// TIA Portal V15.1 export
// export: Created 2026-01-15T16:29:41.881654Z, ExportSetting WithDefaults, WithReadOnly, DisplayName Totally Integrated Automation Portal, DisplayVersion V15.1 Update 8, DisplayName TIA Portal Openness, DisplayVersion V15.1 Update 8, DisplayName STEP 7 Professional, DisplayVersion V15.1 Update 8, DisplayName WinCC Advanced, DisplayVersion V15.1 Update 8
FUNCTION_BLOCK "4.SIMULATION_DATA"   // FB4, LAD
{ S7_Optimized_Access := 'TRUE' }
VERSION : 0.1
// stored: AutoNumber false, CodeModifiedDate 2025-08-27T17:12:03.7644125Z, CompileDate 2026-01-15T16:25:51.5973447Z, CreationDate 2026-01-15T16:22:49.8270549Z, DownloadWithoutReinit false, HandleErrorsWithinBlock false, InterfaceModifiedDate 2023-11-28T22:28:44.2264332Z, IsConsistent true, IsIECCheckEnabled false, IsKnowHowProtected false, IsRetainMemResEnabled false, IsWriteProtected false, LibraryConformanceStatus The object is library-conformant., MemoryReserve 100, ModifiedDate 2025-08-27T17:12:03.7644125Z, ParameterModified 2023-11-28T22:28:44.2264332Z, PLCSimAdvancedSupport false, SetENOAutomatically False, StructureModified 2023-11-28T22:28:44.2264332Z, UDAEnableTagReadback false
   VAR_INPUT
      RE_SET : Bool;
      XUNG_CLOCK : Bool;
      CAN_1 : Bool;
      CAN_2 : Bool;
      CAN_3 : Bool;
      CAN_4 : Bool;
      CAN_5 : Bool;
      CAN_6 : Bool;
      CAN_7 : Bool;
      CAN_8 : Bool;
      CAN_9 : Bool;
      CAN_10 : Bool;
      CAN_11 : Bool;
      CAN_12 : Bool;
      XA_1 : Bool;
      XA_2 : Bool;
      XA_3 : Bool;
      XA_4 : Bool;
      XA_5 : Bool;
      XA_6 : Bool;
      XA_7 : Bool;
      XA_8 : Bool;
      XA_9 : Bool;
      XA_10 : Bool;
      XA_11 : Bool;
      XA_12 : Bool;
      HS_NAP_AGG1 : Real;
      HS_NAP_AGG2 : Real;
      HS_NAP_AGG3 : Real;
      HS_NAP_AGG4 : Real;
      HS_NAP_AGG5 : Real;
      HS_NAP_AGG6 : Real;
      HS_NAP_CEM1 : Real;
      HS_NAP_CEM2 : Real;
      HS_NAP_WAT1 : Real;
      HS_NAP_WAT2 : Real;
      HS_NAP_ADD1 : Real;
      HS_NAP_ADD2 : Real;
      HS_XA_AGG1 : Real;
      HS_XA_AGG2 : Real;
      HS_XA_AGG3 : Real;
      HS_XA_AGG4 : Real;
      HS_XA_AGG5 : Real;
      HS_XA_AGG6 : Real;
      HS_XA_CEM1 : Real;
      HS_XA_CEM2 : Real;
      HS_XA_WAT1 : Real;
      HS_XA_WAT2 : Real;
      HS_XA_ADD1 : Real;
      HS_XA_ADD2 : Real;
   END_VAR
   VAR_OUTPUT
      AGG1 : Real;
      AGG2 : Real;
      AGG3 : Real;
      AGG4 : Real;
      AGG5 : Real;
      AGG6 : Real;
      CEM1 : Real;
      CEM2 : Real;
      WAT1 : Real;
      WAT2 : Real;
      WADD1 : Real;
      WADD2 : Real;
   END_VAR
   VAR
      A1 : Bool;
      B1 : Bool;
      A2 : Bool;
      B2 : Bool;
      A3 : Bool;
      B3 : Bool;
      A4 : Bool;
      B4 : Bool;
      A5 : Bool;
      B5 : Bool;
      A6 : Bool;
      B6 : Bool;
      A7 : Bool;
      B7 : Bool;
      A8 : Bool;
      B8 : Bool;
      A9 : Bool;
      B9 : Bool;
      A10 : Bool;
      B10 : Bool;
      A11 : Bool;
      B11 : Bool;
      A12 : Bool;
      B12 : Bool;
   END_VAR
   VAR_TEMP   // added for the SCL form of the ladder/FBD networks
      _w1 : Bool;
      _w2 : Bool;
   END_VAR
BEGIN

REGION Network 1: RESET
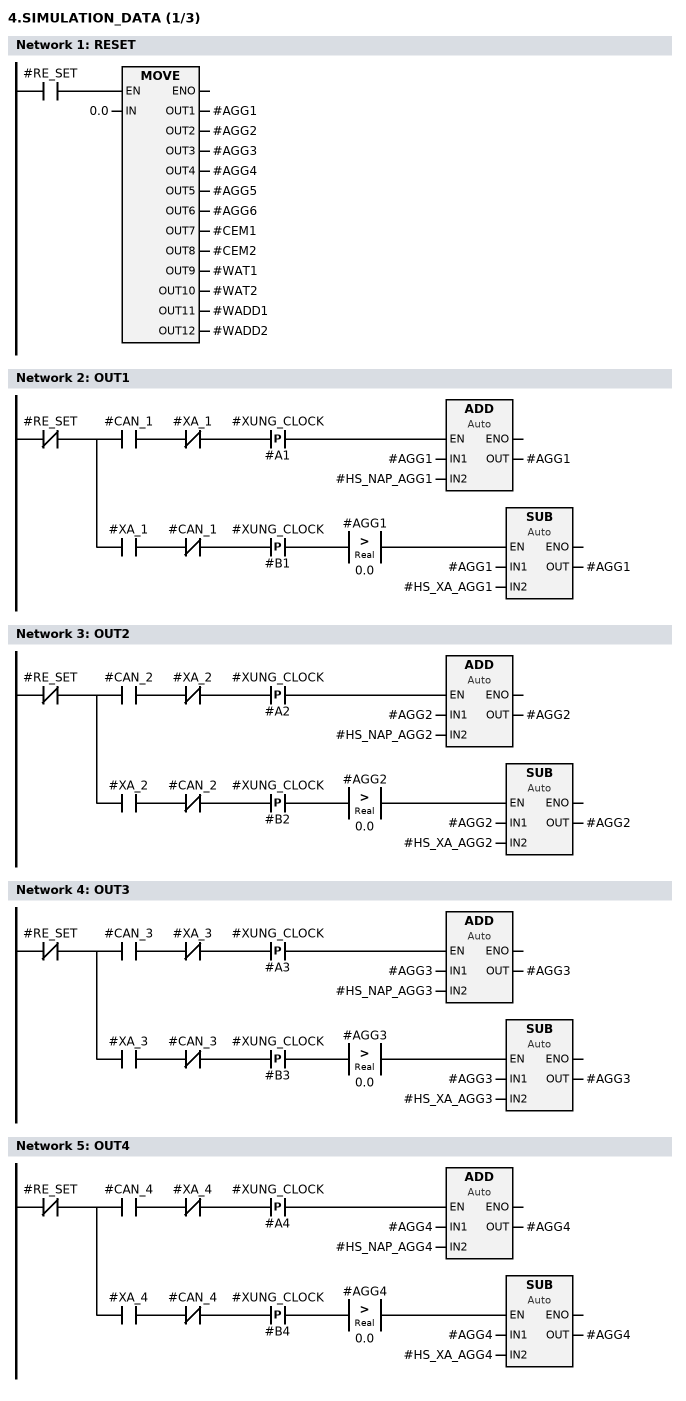
   RUNG wire#powerrail
      Contact( #RE_SET )
      Move(in := 0.0, out1 => #AGG1, out2 => #AGG2, out3 => #AGG3, out4 => #AGG4, out5 => #AGG5, out6 => #AGG6, out7 => #CEM1, out8 => #CEM2, out9 => #WAT1, out10 => #WAT2, out11 => #WADD1, out12 => #WADD2)
   END_RUNG
   // the same network as SCL:
   IF #RE_SET THEN
       #AGG1 := 0.0;
       #AGG2 := 0.0;
       #AGG3 := 0.0;
       #AGG4 := 0.0;
       #AGG5 := 0.0;
       #AGG6 := 0.0;
       #CEM1 := 0.0;
       #CEM2 := 0.0;
       #WAT1 := 0.0;
       #WAT2 := 0.0;
       #WADD1 := 0.0;
       #WADD2 := 0.0;
   END_IF;
END_REGION

REGION Network 2: OUT1
   RUNG wire#powerrail
      I_Contact( #RE_SET )
      wire#w1
      Contact( #CAN_1 )
      I_Contact( #XA_1 )
      P_Contact(operand := #XUNG_CLOCK, bit := #A1)
      Add(in1 := #AGG1, in2 := #HS_NAP_AGG1, out => #AGG1)
   END_RUNG
   RUNG wire#w1
      Contact( #XA_1 )
      I_Contact( #CAN_1 )
      P_Contact(operand := #XUNG_CLOCK, bit := #B1)
      { S7_Templates := "SrcType := Real" } GT_Contact(in1 := #AGG1, in2 := 0.0)
      Sub(in1 := #AGG1, in2 := #HS_XA_AGG1, out => #AGG1)
   END_RUNG
   // the same network as SCL:
   #_w1 := NOT #RE_SET AND #CAN_1 AND NOT #XA_1 AND #XUNG_CLOCK AND NOT #A1;   // rising edge of #XUNG_CLOCK
   #A1 := #XUNG_CLOCK;
   IF #_w1 THEN #AGG1 := #AGG1 + #HS_NAP_AGG1; END_IF;
   #_w2 := NOT #RE_SET AND #XA_1 AND NOT #CAN_1 AND #XUNG_CLOCK AND NOT #B1;   // rising edge of #XUNG_CLOCK
   #B1 := #XUNG_CLOCK;
   IF #_w2 AND (#AGG1 > 0.0) THEN #AGG1 := #AGG1 - #HS_XA_AGG1; END_IF;
END_REGION

REGION Network 3: OUT2
   RUNG wire#powerrail
      I_Contact( #RE_SET )
      wire#w1
      Contact( #CAN_2 )
      I_Contact( #XA_2 )
      P_Contact(operand := #XUNG_CLOCK, bit := #A2)
      Add(in1 := #AGG2, in2 := #HS_NAP_AGG2, out => #AGG2)
   END_RUNG
   RUNG wire#w1
      Contact( #XA_2 )
      I_Contact( #CAN_2 )
      P_Contact(operand := #XUNG_CLOCK, bit := #B2)
      { S7_Templates := "SrcType := Real" } GT_Contact(in1 := #AGG2, in2 := 0.0)
      Sub(in1 := #AGG2, in2 := #HS_XA_AGG2, out => #AGG2)
   END_RUNG
   // the same network as SCL:
   #_w1 := NOT #RE_SET AND #CAN_2 AND NOT #XA_2 AND #XUNG_CLOCK AND NOT #A2;   // rising edge of #XUNG_CLOCK
   #A2 := #XUNG_CLOCK;
   IF #_w1 THEN #AGG2 := #AGG2 + #HS_NAP_AGG2; END_IF;
   #_w2 := NOT #RE_SET AND #XA_2 AND NOT #CAN_2 AND #XUNG_CLOCK AND NOT #B2;   // rising edge of #XUNG_CLOCK
   #B2 := #XUNG_CLOCK;
   IF #_w2 AND (#AGG2 > 0.0) THEN #AGG2 := #AGG2 - #HS_XA_AGG2; END_IF;
END_REGION

REGION Network 4: OUT3
   RUNG wire#powerrail
      I_Contact( #RE_SET )
      wire#w1
      Contact( #CAN_3 )
      I_Contact( #XA_3 )
      P_Contact(operand := #XUNG_CLOCK, bit := #A3)
      Add(in1 := #AGG3, in2 := #HS_NAP_AGG3, out => #AGG3)
   END_RUNG
   RUNG wire#w1
      Contact( #XA_3 )
      I_Contact( #CAN_3 )
      P_Contact(operand := #XUNG_CLOCK, bit := #B3)
      { S7_Templates := "SrcType := Real" } GT_Contact(in1 := #AGG3, in2 := 0.0)
      Sub(in1 := #AGG3, in2 := #HS_XA_AGG3, out => #AGG3)
   END_RUNG
   // the same network as SCL:
   #_w1 := NOT #RE_SET AND #CAN_3 AND NOT #XA_3 AND #XUNG_CLOCK AND NOT #A3;   // rising edge of #XUNG_CLOCK
   #A3 := #XUNG_CLOCK;
   IF #_w1 THEN #AGG3 := #AGG3 + #HS_NAP_AGG3; END_IF;
   #_w2 := NOT #RE_SET AND #XA_3 AND NOT #CAN_3 AND #XUNG_CLOCK AND NOT #B3;   // rising edge of #XUNG_CLOCK
   #B3 := #XUNG_CLOCK;
   IF #_w2 AND (#AGG3 > 0.0) THEN #AGG3 := #AGG3 - #HS_XA_AGG3; END_IF;
END_REGION

REGION Network 5: OUT4
   RUNG wire#powerrail
      I_Contact( #RE_SET )
      wire#w1
      Contact( #CAN_4 )
      I_Contact( #XA_4 )
      P_Contact(operand := #XUNG_CLOCK, bit := #A4)
      Add(in1 := #AGG4, in2 := #HS_NAP_AGG4, out => #AGG4)
   END_RUNG
   RUNG wire#w1
      Contact( #XA_4 )
      I_Contact( #CAN_4 )
      P_Contact(operand := #XUNG_CLOCK, bit := #B4)
      { S7_Templates := "SrcType := Real" } GT_Contact(in1 := #AGG4, in2 := 0.0)
      Sub(in1 := #AGG4, in2 := #HS_XA_AGG4, out => #AGG4)
   END_RUNG
   // the same network as SCL:
   #_w1 := NOT #RE_SET AND #CAN_4 AND NOT #XA_4 AND #XUNG_CLOCK AND NOT #A4;   // rising edge of #XUNG_CLOCK
   #A4 := #XUNG_CLOCK;
   IF #_w1 THEN #AGG4 := #AGG4 + #HS_NAP_AGG4; END_IF;
   #_w2 := NOT #RE_SET AND #XA_4 AND NOT #CAN_4 AND #XUNG_CLOCK AND NOT #B4;   // rising edge of #XUNG_CLOCK
   #B4 := #XUNG_CLOCK;
   IF #_w2 AND (#AGG4 > 0.0) THEN #AGG4 := #AGG4 - #HS_XA_AGG4; END_IF;
END_REGION

REGION Network 6: OUT5
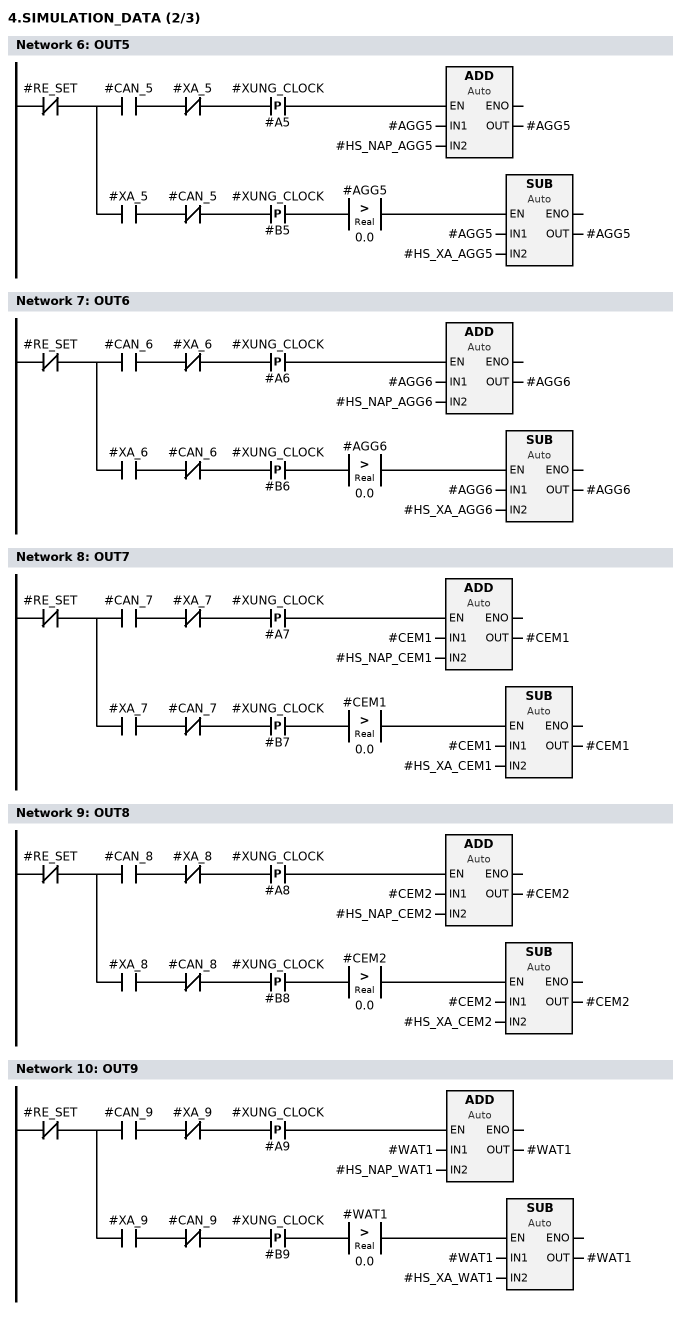
   RUNG wire#powerrail
      I_Contact( #RE_SET )
      wire#w1
      Contact( #CAN_5 )
      I_Contact( #XA_5 )
      P_Contact(operand := #XUNG_CLOCK, bit := #A5)
      Add(in1 := #AGG5, in2 := #HS_NAP_AGG5, out => #AGG5)
   END_RUNG
   RUNG wire#w1
      Contact( #XA_5 )
      I_Contact( #CAN_5 )
      P_Contact(operand := #XUNG_CLOCK, bit := #B5)
      { S7_Templates := "SrcType := Real" } GT_Contact(in1 := #AGG5, in2 := 0.0)
      Sub(in1 := #AGG5, in2 := #HS_XA_AGG5, out => #AGG5)
   END_RUNG
   // the same network as SCL:
   #_w1 := NOT #RE_SET AND #CAN_5 AND NOT #XA_5 AND #XUNG_CLOCK AND NOT #A5;   // rising edge of #XUNG_CLOCK
   #A5 := #XUNG_CLOCK;
   IF #_w1 THEN #AGG5 := #AGG5 + #HS_NAP_AGG5; END_IF;
   #_w2 := NOT #RE_SET AND #XA_5 AND NOT #CAN_5 AND #XUNG_CLOCK AND NOT #B5;   // rising edge of #XUNG_CLOCK
   #B5 := #XUNG_CLOCK;
   IF #_w2 AND (#AGG5 > 0.0) THEN #AGG5 := #AGG5 - #HS_XA_AGG5; END_IF;
END_REGION

REGION Network 7: OUT6
   RUNG wire#powerrail
      I_Contact( #RE_SET )
      wire#w1
      Contact( #CAN_6 )
      I_Contact( #XA_6 )
      P_Contact(operand := #XUNG_CLOCK, bit := #A6)
      Add(in1 := #AGG6, in2 := #HS_NAP_AGG6, out => #AGG6)
   END_RUNG
   RUNG wire#w1
      Contact( #XA_6 )
      I_Contact( #CAN_6 )
      P_Contact(operand := #XUNG_CLOCK, bit := #B6)
      { S7_Templates := "SrcType := Real" } GT_Contact(in1 := #AGG6, in2 := 0.0)
      Sub(in1 := #AGG6, in2 := #HS_XA_AGG6, out => #AGG6)
   END_RUNG
   // the same network as SCL:
   #_w1 := NOT #RE_SET AND #CAN_6 AND NOT #XA_6 AND #XUNG_CLOCK AND NOT #A6;   // rising edge of #XUNG_CLOCK
   #A6 := #XUNG_CLOCK;
   IF #_w1 THEN #AGG6 := #AGG6 + #HS_NAP_AGG6; END_IF;
   #_w2 := NOT #RE_SET AND #XA_6 AND NOT #CAN_6 AND #XUNG_CLOCK AND NOT #B6;   // rising edge of #XUNG_CLOCK
   #B6 := #XUNG_CLOCK;
   IF #_w2 AND (#AGG6 > 0.0) THEN #AGG6 := #AGG6 - #HS_XA_AGG6; END_IF;
END_REGION

REGION Network 8: OUT7
   RUNG wire#powerrail
      I_Contact( #RE_SET )
      wire#w1
      Contact( #CAN_7 )
      I_Contact( #XA_7 )
      P_Contact(operand := #XUNG_CLOCK, bit := #A7)
      Add(in1 := #CEM1, in2 := #HS_NAP_CEM1, out => #CEM1)
   END_RUNG
   RUNG wire#w1
      Contact( #XA_7 )
      I_Contact( #CAN_7 )
      P_Contact(operand := #XUNG_CLOCK, bit := #B7)
      { S7_Templates := "SrcType := Real" } GT_Contact(in1 := #CEM1, in2 := 0.0)
      Sub(in1 := #CEM1, in2 := #HS_XA_CEM1, out => #CEM1)
   END_RUNG
   // the same network as SCL:
   #_w1 := NOT #RE_SET AND #CAN_7 AND NOT #XA_7 AND #XUNG_CLOCK AND NOT #A7;   // rising edge of #XUNG_CLOCK
   #A7 := #XUNG_CLOCK;
   IF #_w1 THEN #CEM1 := #CEM1 + #HS_NAP_CEM1; END_IF;
   #_w2 := NOT #RE_SET AND #XA_7 AND NOT #CAN_7 AND #XUNG_CLOCK AND NOT #B7;   // rising edge of #XUNG_CLOCK
   #B7 := #XUNG_CLOCK;
   IF #_w2 AND (#CEM1 > 0.0) THEN #CEM1 := #CEM1 - #HS_XA_CEM1; END_IF;
END_REGION

REGION Network 9: OUT8
   RUNG wire#powerrail
      I_Contact( #RE_SET )
      wire#w1
      Contact( #CAN_8 )
      I_Contact( #XA_8 )
      P_Contact(operand := #XUNG_CLOCK, bit := #A8)
      Add(in1 := #CEM2, in2 := #HS_NAP_CEM2, out => #CEM2)
   END_RUNG
   RUNG wire#w1
      Contact( #XA_8 )
      I_Contact( #CAN_8 )
      P_Contact(operand := #XUNG_CLOCK, bit := #B8)
      { S7_Templates := "SrcType := Real" } GT_Contact(in1 := #CEM2, in2 := 0.0)
      Sub(in1 := #CEM2, in2 := #HS_XA_CEM2, out => #CEM2)
   END_RUNG
   // the same network as SCL:
   #_w1 := NOT #RE_SET AND #CAN_8 AND NOT #XA_8 AND #XUNG_CLOCK AND NOT #A8;   // rising edge of #XUNG_CLOCK
   #A8 := #XUNG_CLOCK;
   IF #_w1 THEN #CEM2 := #CEM2 + #HS_NAP_CEM2; END_IF;
   #_w2 := NOT #RE_SET AND #XA_8 AND NOT #CAN_8 AND #XUNG_CLOCK AND NOT #B8;   // rising edge of #XUNG_CLOCK
   #B8 := #XUNG_CLOCK;
   IF #_w2 AND (#CEM2 > 0.0) THEN #CEM2 := #CEM2 - #HS_XA_CEM2; END_IF;
END_REGION

REGION Network 10: OUT9
   RUNG wire#powerrail
      I_Contact( #RE_SET )
      wire#w1
      Contact( #CAN_9 )
      I_Contact( #XA_9 )
      P_Contact(operand := #XUNG_CLOCK, bit := #A9)
      Add(in1 := #WAT1, in2 := #HS_NAP_WAT1, out => #WAT1)
   END_RUNG
   RUNG wire#w1
      Contact( #XA_9 )
      I_Contact( #CAN_9 )
      P_Contact(operand := #XUNG_CLOCK, bit := #B9)
      { S7_Templates := "SrcType := Real" } GT_Contact(in1 := #WAT1, in2 := 0.0)
      Sub(in1 := #WAT1, in2 := #HS_XA_WAT1, out => #WAT1)
   END_RUNG
   // the same network as SCL:
   #_w1 := NOT #RE_SET AND #CAN_9 AND NOT #XA_9 AND #XUNG_CLOCK AND NOT #A9;   // rising edge of #XUNG_CLOCK
   #A9 := #XUNG_CLOCK;
   IF #_w1 THEN #WAT1 := #WAT1 + #HS_NAP_WAT1; END_IF;
   #_w2 := NOT #RE_SET AND #XA_9 AND NOT #CAN_9 AND #XUNG_CLOCK AND NOT #B9;   // rising edge of #XUNG_CLOCK
   #B9 := #XUNG_CLOCK;
   IF #_w2 AND (#WAT1 > 0.0) THEN #WAT1 := #WAT1 - #HS_XA_WAT1; END_IF;
END_REGION

REGION Network 11: OUT10
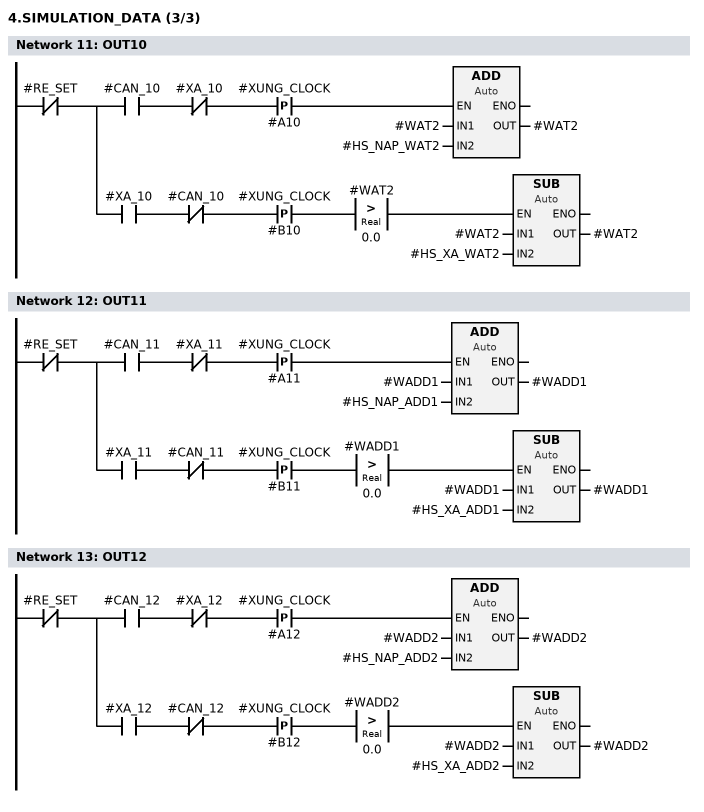
   RUNG wire#powerrail
      I_Contact( #RE_SET )
      wire#w1
      Contact( #CAN_10 )
      I_Contact( #XA_10 )
      P_Contact(operand := #XUNG_CLOCK, bit := #A10)
      Add(in1 := #WAT2, in2 := #HS_NAP_WAT2, out => #WAT2)
   END_RUNG
   RUNG wire#w1
      Contact( #XA_10 )
      I_Contact( #CAN_10 )
      P_Contact(operand := #XUNG_CLOCK, bit := #B10)
      { S7_Templates := "SrcType := Real" } GT_Contact(in1 := #WAT2, in2 := 0.0)
      Sub(in1 := #WAT2, in2 := #HS_XA_WAT2, out => #WAT2)
   END_RUNG
   // the same network as SCL:
   #_w1 := NOT #RE_SET AND #CAN_10 AND NOT #XA_10 AND #XUNG_CLOCK AND NOT #A10;   // rising edge of #XUNG_CLOCK
   #A10 := #XUNG_CLOCK;
   IF #_w1 THEN #WAT2 := #WAT2 + #HS_NAP_WAT2; END_IF;
   #_w2 := NOT #RE_SET AND #XA_10 AND NOT #CAN_10 AND #XUNG_CLOCK AND NOT #B10;   // rising edge of #XUNG_CLOCK
   #B10 := #XUNG_CLOCK;
   IF #_w2 AND (#WAT2 > 0.0) THEN #WAT2 := #WAT2 - #HS_XA_WAT2; END_IF;
END_REGION

REGION Network 12: OUT11
   RUNG wire#powerrail
      I_Contact( #RE_SET )
      wire#w1
      Contact( #CAN_11 )
      I_Contact( #XA_11 )
      P_Contact(operand := #XUNG_CLOCK, bit := #A11)
      Add(in1 := #WADD1, in2 := #HS_NAP_ADD1, out => #WADD1)
   END_RUNG
   RUNG wire#w1
      Contact( #XA_11 )
      I_Contact( #CAN_11 )
      P_Contact(operand := #XUNG_CLOCK, bit := #B11)
      { S7_Templates := "SrcType := Real" } GT_Contact(in1 := #WADD1, in2 := 0.0)
      Sub(in1 := #WADD1, in2 := #HS_XA_ADD1, out => #WADD1)
   END_RUNG
   // the same network as SCL:
   #_w1 := NOT #RE_SET AND #CAN_11 AND NOT #XA_11 AND #XUNG_CLOCK AND NOT #A11;   // rising edge of #XUNG_CLOCK
   #A11 := #XUNG_CLOCK;
   IF #_w1 THEN #WADD1 := #WADD1 + #HS_NAP_ADD1; END_IF;
   #_w2 := NOT #RE_SET AND #XA_11 AND NOT #CAN_11 AND #XUNG_CLOCK AND NOT #B11;   // rising edge of #XUNG_CLOCK
   #B11 := #XUNG_CLOCK;
   IF #_w2 AND (#WADD1 > 0.0) THEN #WADD1 := #WADD1 - #HS_XA_ADD1; END_IF;
END_REGION

REGION Network 13: OUT12
   RUNG wire#powerrail
      I_Contact( #RE_SET )
      wire#w1
      Contact( #CAN_12 )
      I_Contact( #XA_12 )
      P_Contact(operand := #XUNG_CLOCK, bit := #A12)
      Add(in1 := #WADD2, in2 := #HS_NAP_ADD2, out => #WADD2)
   END_RUNG
   RUNG wire#w1
      Contact( #XA_12 )
      I_Contact( #CAN_12 )
      P_Contact(operand := #XUNG_CLOCK, bit := #B12)
      { S7_Templates := "SrcType := Real" } GT_Contact(in1 := #WADD2, in2 := 0.0)
      Sub(in1 := #WADD2, in2 := #HS_XA_ADD2, out => #WADD2)
   END_RUNG
   // the same network as SCL:
   #_w1 := NOT #RE_SET AND #CAN_12 AND NOT #XA_12 AND #XUNG_CLOCK AND NOT #A12;   // rising edge of #XUNG_CLOCK
   #A12 := #XUNG_CLOCK;
   IF #_w1 THEN #WADD2 := #WADD2 + #HS_NAP_ADD2; END_IF;
   #_w2 := NOT #RE_SET AND #XA_12 AND NOT #CAN_12 AND #XUNG_CLOCK AND NOT #B12;   // rising edge of #XUNG_CLOCK
   #B12 := #XUNG_CLOCK;
   IF #_w2 AND (#WADD2 > 0.0) THEN #WADD2 := #WADD2 - #HS_XA_ADD2; END_IF;
END_REGION
END_FUNCTION_BLOCK
